TYPE ST_SendDpConfig :
STRUCT
	nDpDpId			 			: UINT := 0;
	fTimeout		 			: REAL := 0.5;
END_STRUCT
END_TYPE

(* stored: Version 1.1.0.1, ProductVersion 3.1.4024.12
   DUT ST_SendDpConfig: Id {f464b77f-746f-0396-2c2c-8681a9bdcae0} *)
